Staubli VAL3: motionStatus.pgx

public program motionStatus(num x_nInConnFlag)
begin

  // update connection status on port 11000 (motion server)

  switch x_nInConnFlag
    case -1
      userPageSet("uxMonitor", "lblMotionState", "innerHTML", "connection lost")
    break
    case 0
      userPageSet("uxMonitor", "lblMotionState", "innerHTML", "not connected")
    break
    case 1
      userPageSet("uxMonitor", "lblMotionState", "innerHTML", "connected")
    break
    default
      userPageSet("uxMonitor", "lblMotionState", "innerHTML", "not connected")
    break
  endSwitch

end
